FUNCTION_BLOCK FB_JetNozzle2
VAR_INPUT
END_VAR
VAR_OUTPUT
END_VAR
VAR
	//Properties
	bError 					: BOOL := FALSE;
	fAngleActual 			: REAL;
	fAngleSetpoint 			: REAL := 50;
	//Raw values
	nAngleActual AT %I*		: INT;
	nAngleSetpoint AT %Q* 	: INT;
END_VAR

PROPERTY AngleActual : REAL
GET
AngleActual := THIS^.fAngleActual;
END_GET
SET
THIS^.fAngleActual := AngleActual;
END_SET
END_PROPERTY

PROPERTY AngleSetpoint : REAL
GET
AngleSetpoint := THIS^.fAngleSetpoint;
END_GET
SET
THIS^.fAngleSetpoint := AngleSetpoint;
END_SET
END_PROPERTY

PROPERTY Error : BOOL
GET
Error := THIS^.bError;
END_GET
SET
THIS^.bError := Error;
END_SET
END_PROPERTY

METHOD Run
VAR_INPUT
END_VAR
//Read feedback for opening position
fAngleActual := FC_Voltage2_10Raw_TO_Percentage(nAngleActual);

//Write setpoint for opening position
nAngleSetpoint := FC_Percentage_TO_Voltage2_10Raw(fAngleSetpoint);
END_METHOD

END_FUNCTION_BLOCK

(* stored: Version 1.1.0.1, ProductVersion 3.1.4024.0
   POU FB_JetNozzle2: Id {5812933b-cab8-4002-bdfb-a7669d9feb5f}, SpecialFunc None
   Property AngleActual: Id {14f03dc7-a61e-460f-a470-c6e6a22fb447}
   Get Get: Id {cbde43a0-23a6-4cc6-9b7c-1883e580da6e}
   Set Set: Id {30a477b6-7501-41e2-9534-9e86af5679fc}
   Property AngleSetpoint: Id {6e580ee8-d0f1-433b-8fc9-f5d39e71c251}
   Get Get: Id {42622766-6952-44e9-b94b-e19474cc1992}
   Set Set: Id {ba6f40da-b997-4399-a96d-d622c86d37be}
   Property Error: Id {2ea5aa42-99dc-4caa-a5e0-eb2913c1c8cd}
   Get Get: Id {9ea0242f-3427-4c66-9b20-2fea983566fb}
   Set Set: Id {9bdf0e08-c9a2-4798-b8dd-01f334df07ba}
   Method Run: Id {566a8166-3349-479f-b942-9ffe250e1651} *)
